// TIA Portal project "projet_iei5_bald_sacewicz" (V17)

(* hardware
DEVICE "S7-1200 station_1"  S7-1200 Station
   slot 0: "Rack_0"  S7-1200 Rack  Rack  V1.0
   slot 1: "PLC_1"  CPU 1214C AC/DC/Rly  6ES7 214-1BE30-0XB0  V2.2
*)

// ===== PLC "PLC_1"  CPU 1214C AC/DC/Rly =====

VAR_GLOBAL   // PLC tag table "Default tag table"
   "LED" AT %Q0.0 : Bool;
   "LED2" AT %Q0.1 : Bool;
   "adrssseAI_potentiometre" AT %IW64 : Word;
   "Tag_2" AT %MD10 : DWord;
   "Tag_1" AT %MD12 : Real;
   "Tag_3" AT %MW14 : Int;
   "Tag_4" AT %M0.1 : Bool;
   "LED3" AT %Q0.2 : Bool;
   "MoteurPin1" AT %Q0.3 : Bool;
   "MoteurPin2" AT %Q0.4 : Bool;
   "MoteurPin3" AT %Q0.5 : Bool;
   "MoteurPin4" AT %Q0.6 : Bool;
   "MoteurMarche" AT %I0.2 : Bool;
   "Memento" AT %M0.5 : Bool;
   "Step1" AT %M0.6 : Bool;
   "Step2" AT %M0.7 : Bool;
   "MoteurMarche2" AT %I0.3 : Bool;
   "MoteurMarche3" AT %I0.4 : Bool;
   "MoteurMarch4" AT %I0.5 : Bool;
   "Step3" AT %M1.0 : Bool;
   "Step4" AT %M1.1 : Bool;
   "interrupteur_gauche" AT %I1.0 : Bool;
   "interrupteur_droite" AT %I1.1 : Bool;
   "step5" AT %M1.2 : Bool;
   "step6" AT %M1.3 : Bool;
   "step7" AT %M1.4 : Bool;
   "step8" AT %M1.5 : Bool;
END_VAR

// folder: System blocks/Program resources

DATA_BLOCK "IEC_Timer_0_DB_4"   // DB5
{ S7_Optimized_Access := 'TRUE' }
AUTHOR : Simatic
FAMILY : IEC
NAME : IEC_TMR
VERSION : 1.0
// stored: InstanceOfName IEC_TIMER
"IEC_TIMER"
BEGIN
END_DATA_BLOCK

DATA_BLOCK "IEC_Timer_0_DB_5"   // DB6
{ S7_Optimized_Access := 'TRUE' }
AUTHOR : Simatic
FAMILY : IEC
NAME : IEC_TMR
VERSION : 1.0
// stored: InstanceOfName IEC_TIMER
"IEC_TIMER"
BEGIN
END_DATA_BLOCK

DATA_BLOCK "IEC_Timer_0_DB_6"   // DB7
{ S7_Optimized_Access := 'TRUE' }
AUTHOR : Simatic
FAMILY : IEC
NAME : IEC_TMR
VERSION : 1.0
// stored: InstanceOfName IEC_TIMER
"IEC_TIMER"
BEGIN
END_DATA_BLOCK

DATA_BLOCK "IEC_Timer_0_DB_7"   // DB8
{ S7_Optimized_Access := 'TRUE' }
AUTHOR : Simatic
FAMILY : IEC
NAME : IEC_TMR
VERSION : 1.0
// stored: InstanceOfName IEC_TIMER
"IEC_TIMER"
BEGIN
END_DATA_BLOCK

DATA_BLOCK "IEC_Timer_0_DB_8"   // DB9
{ S7_Optimized_Access := 'TRUE' }
AUTHOR : Simatic
FAMILY : IEC
NAME : IEC_TMR
VERSION : 1.0
// stored: InstanceOfName IEC_TIMER
"IEC_TIMER"
BEGIN
END_DATA_BLOCK

DATA_BLOCK "IEC_Timer_0_DB_9"   // DB10
{ S7_Optimized_Access := 'TRUE' }
AUTHOR : Simatic
FAMILY : IEC
NAME : IEC_TMR
VERSION : 1.0
// stored: InstanceOfName IEC_TIMER
"IEC_TIMER"
BEGIN
END_DATA_BLOCK

DATA_BLOCK "IEC_Timer_0_DB_10"   // DB11
{ S7_Optimized_Access := 'TRUE' }
AUTHOR : Simatic
FAMILY : IEC
NAME : IEC_TMR
VERSION : 1.0
// stored: InstanceOfName IEC_TIMER
"IEC_TIMER"
BEGIN
END_DATA_BLOCK

DATA_BLOCK "IEC_Timer_0_DB_11"   // DB12
{ S7_Optimized_Access := 'TRUE' }
AUTHOR : Simatic
FAMILY : IEC
NAME : IEC_TMR
VERSION : 1.0
// stored: InstanceOfName IEC_TIMER
"IEC_TIMER"
BEGIN
END_DATA_BLOCK

// folder: (top level)

FUNCTION "Block_1" : Void   // FC1, FBD
{ S7_Optimized_Access := 'TRUE' }
VERSION : 0.1
BEGIN

REGION Network 1
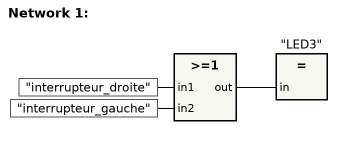
   "LED3" := "interrupteur_droite" OR "interrupteur_gauche";
END_REGION
END_FUNCTION

FUNCTION "poten" : Void   // FC2, LAD
{ S7_Optimized_Access := 'TRUE' }
VERSION : 0.1
BEGIN

REGION Network 1: POTENTIOMETRE
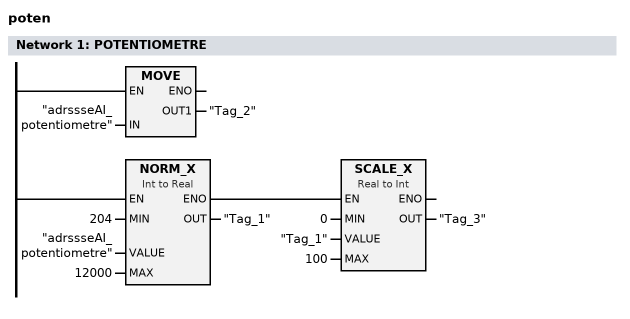
   RUNG wire#powerrail
      { S7_GenerateENO := "TRUE" } Move(in := "adrssseAI_potentiometre", out1 => "Tag_2")
   END_RUNG
   RUNG wire#powerrail
      { S7_Templates := "[SrcType := Int, DestType := Real]"; S7_GenerateENO := "TRUE" } Normalize(min := 204, value := "adrssseAI_potentiometre", max := 12000, out => "Tag_1")
      { S7_Templates := "[SrcType := Real, DestType := Int]"; S7_GenerateENO := "TRUE" } Scale(min := 0, value := "Tag_1", max := 100, out => "Tag_3")
   END_RUNG
   // the same network as SCL:
   // ENO of a box is taken as its EN; it also drops when the box reports an error
   "Tag_2" := "adrssseAI_potentiometre";
   "Tag_1" := NORM_X(MIN := 204, VALUE := "adrssseAI_potentiometre", MAX := 12000);
   "Tag_3" := SCALE_X(MIN := 0, VALUE := "Tag_1", MAX := 100);
END_REGION
END_FUNCTION

FUNCTION "moteur_man" : Void   // FC4, FBD
{ S7_Optimized_Access := 'TRUE' }
VERSION : 0.1
   VAR_TEMP   // added for the SCL form of the ladder/FBD networks
      _w1 : Bool;
   END_VAR
BEGIN

REGION Network 1
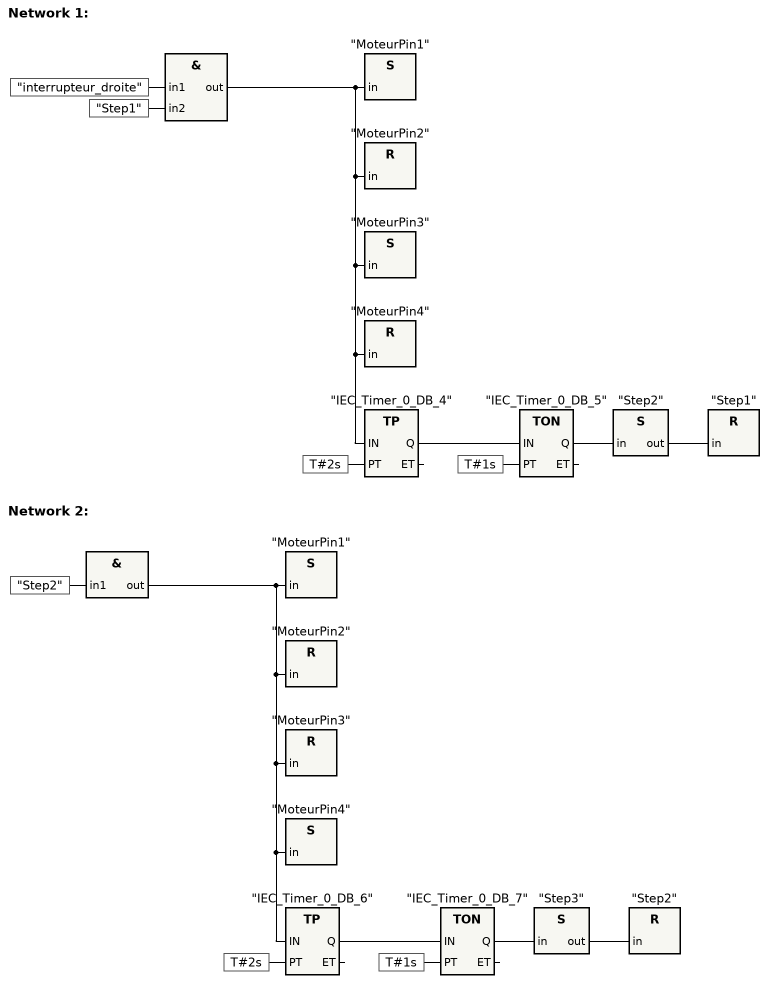
   #_w1 := "interrupteur_droite" AND "Step1";
   IF #_w1 THEN
       "MoteurPin1" := TRUE;
       "MoteurPin2" := FALSE;
       "MoteurPin3" := TRUE;
       "MoteurPin4" := FALSE;
   END_IF;
   "IEC_Timer_0_DB_4".TP(IN := #_w1, PT := T#2s);
   "IEC_Timer_0_DB_5".TON(IN := "IEC_Timer_0_DB_4".Q, PT := T#1s);
   IF "IEC_Timer_0_DB_5".Q THEN
       "Step2" := TRUE;
       "Step1" := FALSE;
   END_IF;
END_REGION

REGION Network 2
   IF "Step2" THEN
       "MoteurPin1" := TRUE;
       "MoteurPin2" := FALSE;
       "MoteurPin3" := FALSE;
       "MoteurPin4" := TRUE;
   END_IF;
   "IEC_Timer_0_DB_6".TP(IN := "Step2", PT := T#2s);
   "IEC_Timer_0_DB_7".TON(IN := "IEC_Timer_0_DB_6".Q, PT := T#1s);
   IF "IEC_Timer_0_DB_7".Q THEN
       "Step3" := TRUE;
       "Step2" := FALSE;
   END_IF;
END_REGION

REGION Network 3
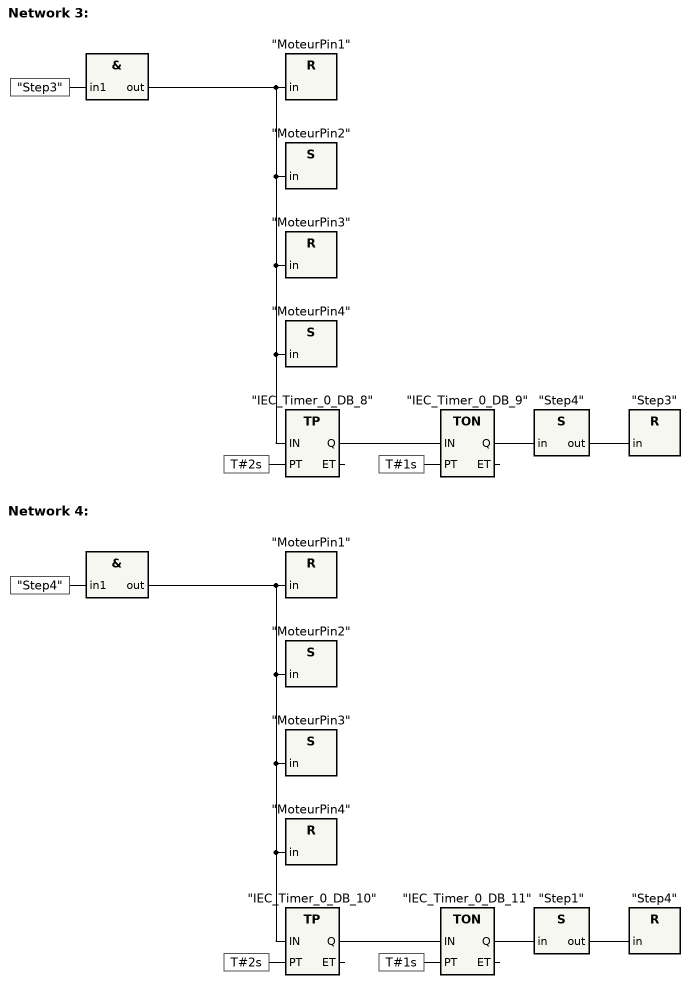
   IF "Step3" THEN
       "MoteurPin1" := FALSE;
       "MoteurPin2" := TRUE;
       "MoteurPin3" := FALSE;
       "MoteurPin4" := TRUE;
   END_IF;
   "IEC_Timer_0_DB_8".TP(IN := "Step3", PT := T#2s);
   "IEC_Timer_0_DB_9".TON(IN := "IEC_Timer_0_DB_8".Q, PT := T#1s);
   IF "IEC_Timer_0_DB_9".Q THEN
       "Step4" := TRUE;
       "Step3" := FALSE;
   END_IF;
END_REGION

REGION Network 4
   IF "Step4" THEN
       "MoteurPin1" := FALSE;
       "MoteurPin2" := TRUE;
       "MoteurPin3" := TRUE;
       "MoteurPin4" := FALSE;
   END_IF;
   "IEC_Timer_0_DB_10".TP(IN := "Step4", PT := T#2s);
   "IEC_Timer_0_DB_11".TON(IN := "IEC_Timer_0_DB_10".Q, PT := T#1s);
   IF "IEC_Timer_0_DB_11".Q THEN
       "Step1" := TRUE;
       "Step4" := FALSE;
   END_IF;
END_REGION

REGION Network 5: moteur inverse
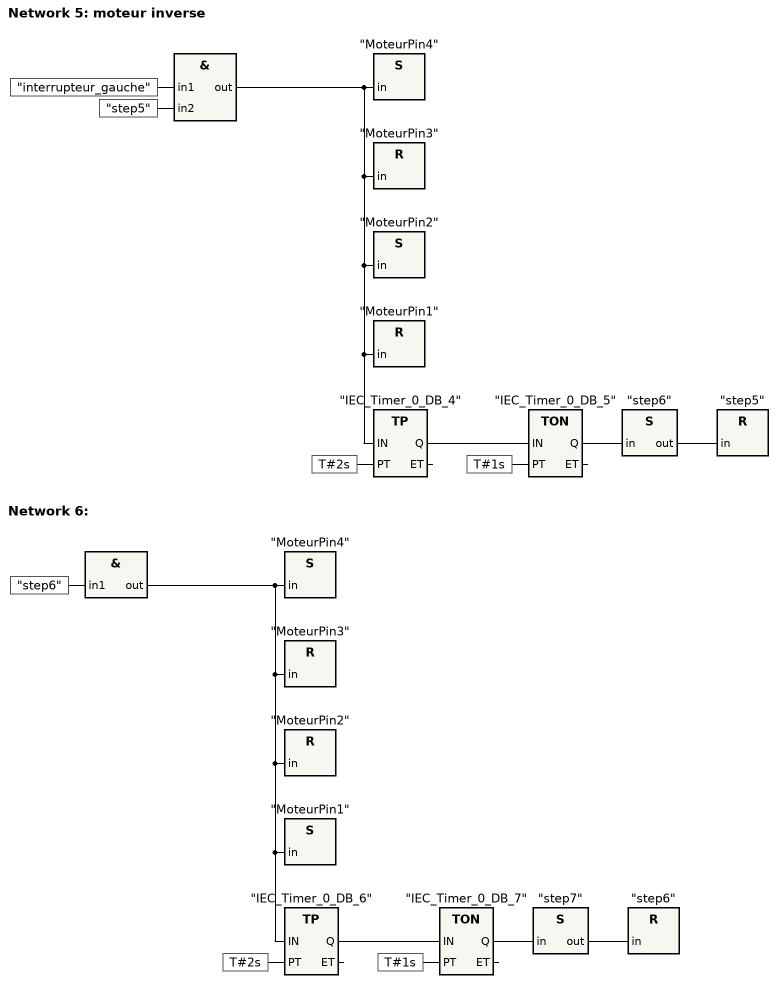
   #_w1 := "interrupteur_gauche" AND "step5";
   IF #_w1 THEN
       "MoteurPin4" := TRUE;
       "MoteurPin3" := FALSE;
       "MoteurPin2" := TRUE;
       "MoteurPin1" := FALSE;
   END_IF;
   "IEC_Timer_0_DB_4".TP(IN := #_w1, PT := T#2s);
   "IEC_Timer_0_DB_5".TON(IN := "IEC_Timer_0_DB_4".Q, PT := T#1s);
   IF "IEC_Timer_0_DB_5".Q THEN
       "step6" := TRUE;
       "step5" := FALSE;
   END_IF;
END_REGION

REGION Network 6
   IF "step6" THEN
       "MoteurPin4" := TRUE;
       "MoteurPin3" := FALSE;
       "MoteurPin2" := FALSE;
       "MoteurPin1" := TRUE;
   END_IF;
   "IEC_Timer_0_DB_6".TP(IN := "step6", PT := T#2s);
   "IEC_Timer_0_DB_7".TON(IN := "IEC_Timer_0_DB_6".Q, PT := T#1s);
   IF "IEC_Timer_0_DB_7".Q THEN
       "step7" := TRUE;
       "step6" := FALSE;
   END_IF;
END_REGION

REGION Network 7
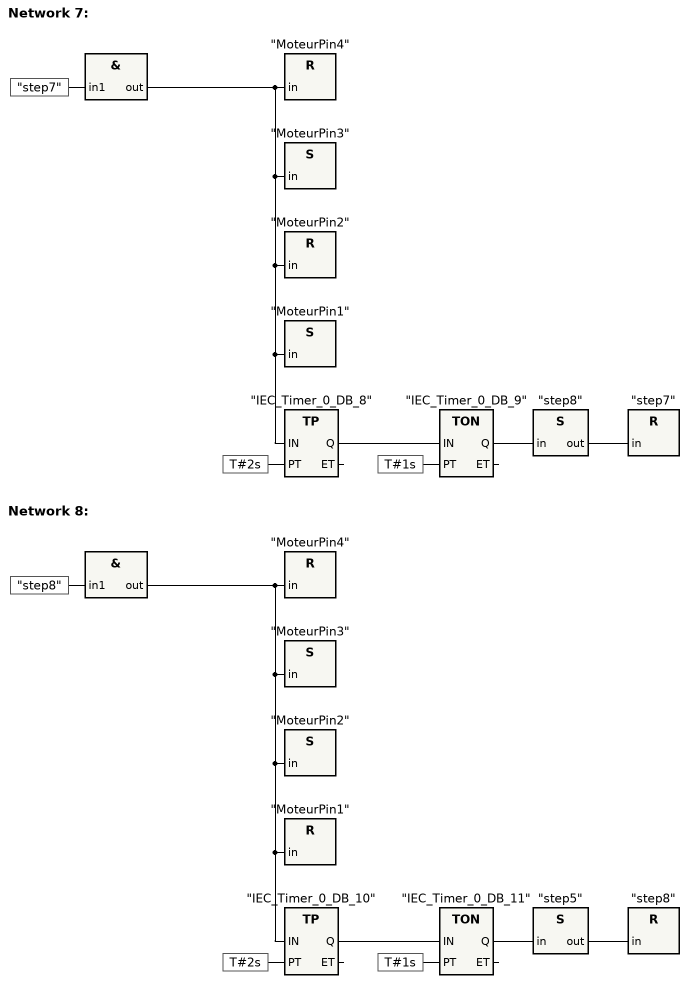
   IF "step7" THEN
       "MoteurPin4" := FALSE;
       "MoteurPin3" := TRUE;
       "MoteurPin2" := FALSE;
       "MoteurPin1" := TRUE;
   END_IF;
   "IEC_Timer_0_DB_8".TP(IN := "step7", PT := T#2s);
   "IEC_Timer_0_DB_9".TON(IN := "IEC_Timer_0_DB_8".Q, PT := T#1s);
   IF "IEC_Timer_0_DB_9".Q THEN
       "step8" := TRUE;
       "step7" := FALSE;
   END_IF;
END_REGION

REGION Network 8
   IF "step8" THEN
       "MoteurPin4" := FALSE;
       "MoteurPin3" := TRUE;
       "MoteurPin2" := TRUE;
       "MoteurPin1" := FALSE;
   END_IF;
   "IEC_Timer_0_DB_10".TP(IN := "step8", PT := T#2s);
   "IEC_Timer_0_DB_11".TON(IN := "IEC_Timer_0_DB_10".Q, PT := T#1s);
   IF "IEC_Timer_0_DB_11".Q THEN
       "step5" := TRUE;
       "step8" := FALSE;
   END_IF;
END_REGION
END_FUNCTION

ORGANIZATION_BLOCK "Main"   // OB1, LAD, ProgramCycle
TITLE = "Main Program Sweep (Cycle)"
{ S7_Optimized_Access := 'TRUE' }
VERSION : 0.1
BEGIN

REGION Network 1
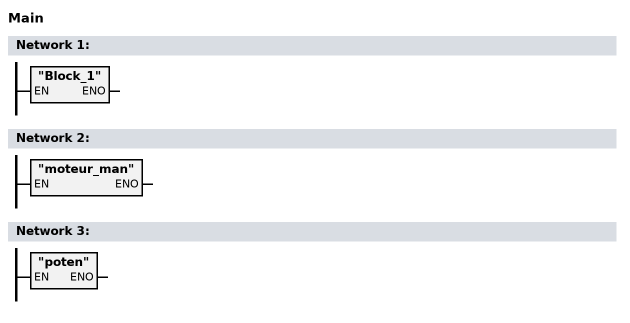
   RUNG wire#powerrail
      "Block_1"()
   END_RUNG
   // the same network as SCL:
   "Block_1"();
END_REGION

REGION Network 2
   RUNG wire#powerrail
      "moteur_man"()
   END_RUNG
   // the same network as SCL:
   "moteur_man"();
END_REGION

REGION Network 3
   RUNG wire#powerrail
      "poten"()
   END_RUNG
   // the same network as SCL:
   "poten"();
END_REGION
END_ORGANIZATION_BLOCK

ORGANIZATION_BLOCK "Startup"   // OB100, FBD, Startup
TITLE = "Complete Restart"
{ S7_Optimized_Access := 'TRUE' }
VERSION : 0.1
   VAR_INPUT
      LostRetentive : Bool;   // True if retentive data are lost
      LostRTC : Bool;   // True if date and time are lost
   END_VAR
BEGIN

REGION Network 1
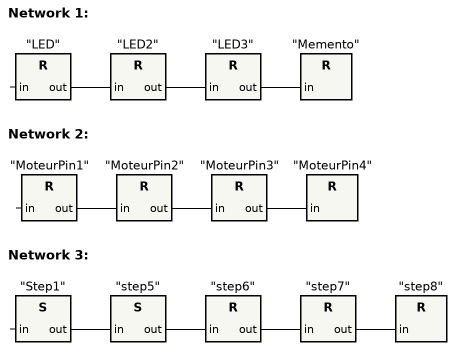
   "LED" := FALSE;
   "LED2" := FALSE;
   "LED3" := FALSE;
   "Memento" := FALSE;
END_REGION

REGION Network 2
   "MoteurPin1" := FALSE;
   "MoteurPin2" := FALSE;
   "MoteurPin3" := FALSE;
   "MoteurPin4" := FALSE;
END_REGION

REGION Network 3
   "Step1" := TRUE;
   "step5" := TRUE;
   "step6" := FALSE;
   "step7" := FALSE;
   "step8" := FALSE;
END_REGION
END_ORGANIZATION_BLOCK